// TIA Portal V20 export
// export: Created 2025-12-01T14:57:40.6788233Z, ExportSetting None, DisplayName Totally Integrated Automation Portal, DisplayVersion V20 Update 3, DisplayName TIA Portal Openness, DisplayVersion V20 Update 3, DisplayName TIA Portal Version Control Interface, DisplayVersion V20 Update 3, DisplayName STEP 7 Professional, DisplayVersion V20 Update 3, DisplayName STEP 7 Safety, DisplayVersion V20 Update 2, DisplayName WinCC Basic/Comfort/Advanced, DisplayVersion V20 Update 3, DisplayName WinCC Professional, DisplayVersion V20 Update 3, DisplayName WinCC Unified, DisplayVersion V20 Update 3
FUNCTION_BLOCK "FB291_M_CIMCORP_Descarga_Doble"   // FB291, LAD
TITLE = M_TRANSLO_CS_DESCARGA_E0_S3
{ S7_Optimized_Access := 'FALSE' }
AUTHOR : CIMCORP
NAME : 20160509
VERSION : 3.4
// stored: AutoNumber false, SetENOAutomatically false
   VAR_INPUT
      Mesa : UInt;   // Mesa de la FB
      Error_Tx : Bool;   // Error en el Tx
      EnTension : Bool;   // Existe Tension en la Mesa
      Termico_Tx : Bool;   // Proteccion del Tx
      pHsMx_P1 : Bool;   // pHs 1 de la Mesa
      pHsMx_P2 : Bool;   // pHs 2 de la Mesa
      pHsMx_Seg : Bool;   // pHs Seguridad de la Mesa
      Avance_Tx : Bool;   // Avance del Tx
      CIMCORP_MoveOK_P1 : Bool;   // CIMCORP >> Move OK P01
      CIMCORP_MoveOK_P2 : Bool;   // CIMCORP >> Move OK P02
      CIMCORP_Stop : Bool;   // CIMCORP >> Stop
      PTF_Mx_MSig : Bool;   // S3 >> Mesa Siguiente PTF
      FTF_Mx_MSig : Bool;   // S3 >> Mesa Siguiente FTF
      MSig_CargaAct : Bool;
      Mx_VelocidadLenta_In : Bool;   // Forzar a Velociada Lenta
      F_EnvMens_Mx : Bool;   // Fin de Envio de Mensaje
      OrdSal_S03 : Bool;   // Orden de Salida por S3
      V_CNT_ApHsMx : Int := 200;   // Valor de Ausencia
      V_CNTSeg_ApHsMx : Int := 2000;   // Valor de Seguriadad para Ausencia
      V_CNT_PerdidapHs : Int := 1000;   // CNT de Perdida de pHs
   END_VAR
   VAR_OUTPUT
      P_EnvMens_PMx : Bool;   // Permiso de Enviar Mensaje de Presencia
      P_RecepOK_Mx : Bool;   // Recepcion OK
      AVTF_Mx_MSig : Bool;   // S3 >> Mesa Siguiente AVTF
      P_Mens_Mx_MSig : Bool;   // S3 >> Mesa Siguiente P_Mens
   END_VAR
   VAR
      Mx_ET00 : Bool;
      Mx_ET01 : Bool;
      Mx_ET02 : Bool;
      Mx_ET06 : Bool;
      Mx_ET07 : Bool;
      Mx_ET08 : Bool;
      Mx_ET09 : Bool;
      Mx_ET10 : Bool;
      Mx_ET11 : Bool;
      Mx_ET110 : Bool;
      Mx_ET111 : Bool;
      Mx_ET20 : Bool;
      Mx_ET21 : Bool;
      Mx_ET120 : Bool;
      Mx_ET121 : Bool;
      Mx_ET50 : Bool;
      Mx_ET51 : Bool;
      Mx_ET150 : Bool;
      Mx_ET151 : Bool;
      CIMCORP_OK : Bool;   // CIMCORP >> Esta En Marcha
      CNT_ApHsMx { S7_SetPoint := 'True'} : "FB910_CNT_UHS";   // CNT de la Ausencia
      CNTSeg_ApHsMx { S7_SetPoint := 'True'} : "FB910_CNT_UHS";   // CNT de Seguridad de la Ausencia
      TMP_EnTension { S7_SetPoint := 'True'} : "FB910_CNT_UHS";
      CNT_PerdidapHs { S7_SetPoint := 'True'} : "FB910_CNT_UHS";   // CNT de Perdida de pHs
      STAT_EnvMens_PMx : Bool;   // Interna >> Envio del Mensaje de Presencia
      STAT_AVTF_Mx_MSig : Bool;   // Interna >> AVTF de Mx >> MSig
      MA_UnLoadOK_P1 : Bool;
      MA_UnLoadOK_P2 : Bool;
   END_VAR
   VAR_TEMP
      EstadoZona : "EstadoZona";   // Estado de Zona de la Mesa
      EstadoVI : "EstadosMesa";   // Estado del Vehiculo Inteliguente de la Mesa
      ConfigFB : "UDT_ConfigFB";   // Configuracion de la FB de la Mesa
      Aux_ET00 : Bool;
   END_VAR
BEGIN

REGION Network 1: INICIALIZAR - Recoger las Variables de Estado de la Mesa
   // Se recoge - Estado_CBx
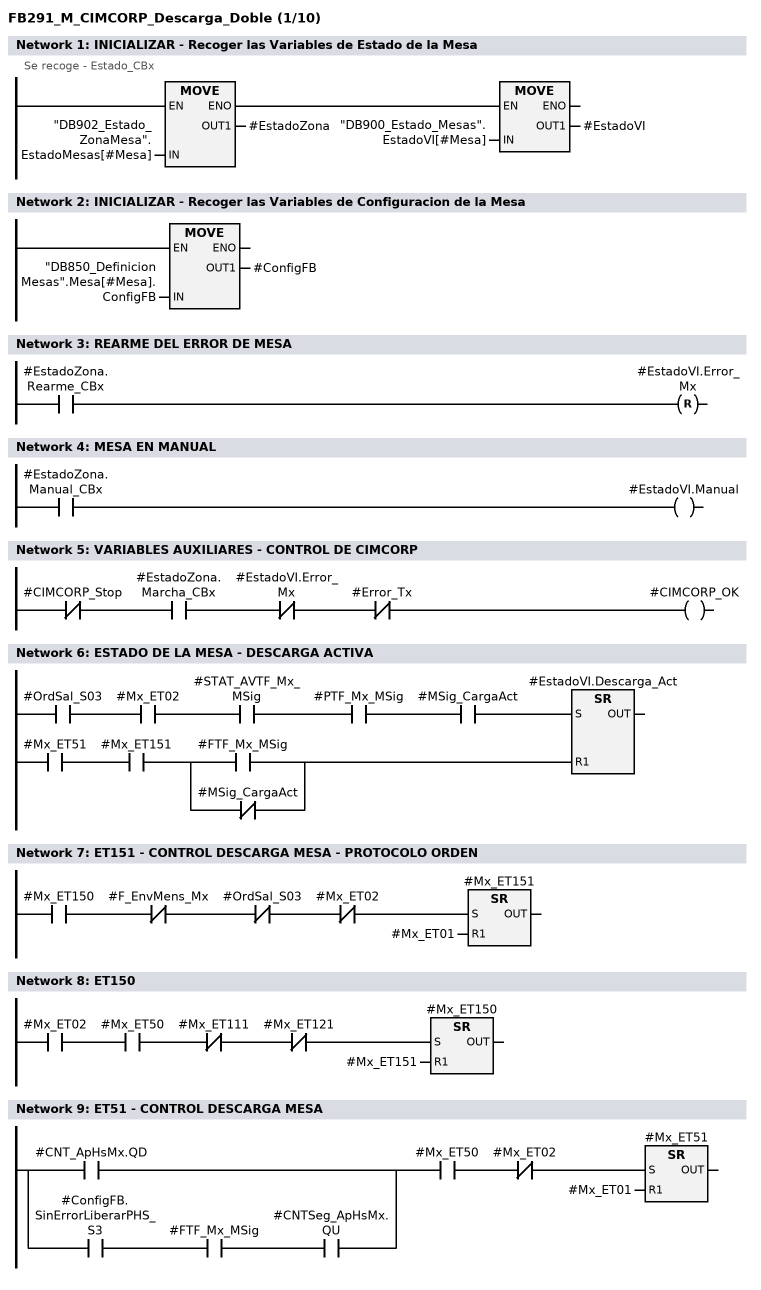
   RUNG wire#powerrail
      Move(in := "DB902_Estado_ZonaMesa".EstadoMesas[#Mesa], out1 => #EstadoZona)
      Move(in := "DB900_Estado_Mesas".EstadoVI[#Mesa], out1 => #EstadoVI)
   END_RUNG
   // the same network as SCL:
   #EstadoZona := "DB902_Estado_ZonaMesa".EstadoMesas[#Mesa];
   #EstadoVI := "DB900_Estado_Mesas".EstadoVI[#Mesa];
END_REGION

REGION Network 2: INICIALIZAR - Recoger las Variables de Configuracion de la Mesa
   RUNG wire#powerrail
      Move(in := "DB850_DefinicionMesas".Mesa[#Mesa].ConfigFB, out1 => #ConfigFB)
   END_RUNG
   // the same network as SCL:
   #ConfigFB := "DB850_DefinicionMesas".Mesa[#Mesa].ConfigFB;
END_REGION

REGION Network 3: REARME DEL ERROR DE MESA
   RUNG wire#powerrail
      Contact( #EstadoZona.Rearme_CBx )
      R_Coil( #EstadoVI.Error_Mx )
   END_RUNG
   // the same network as SCL:
   IF #EstadoZona.Rearme_CBx THEN #EstadoVI.Error_Mx := FALSE; END_IF;
END_REGION

REGION Network 4: MESA EN MANUAL
   RUNG wire#powerrail
      Contact( #EstadoZona.Manual_CBx )
      Coil( #EstadoVI.Manual )
   END_RUNG
   // the same network as SCL:
   #EstadoVI.Manual := #EstadoZona.Manual_CBx;
END_REGION

REGION Network 5: VARIABLES AUXILIARES - CONTROL DE CIMCORP
   RUNG wire#powerrail
      I_Contact( #CIMCORP_Stop )
      Contact( #EstadoZona.Marcha_CBx )
      I_Contact( #EstadoVI.Error_Mx )
      I_Contact( #Error_Tx )
      Coil( #CIMCORP_OK )
   END_RUNG
   // the same network as SCL:
   #CIMCORP_OK := NOT #CIMCORP_Stop AND #EstadoZona.Marcha_CBx AND NOT #EstadoVI.Error_Mx AND NOT #Error_Tx;
END_REGION

REGION Network 6: ESTADO DE LA MESA - DESCARGA ACTIVA
   RUNG wire#powerrail
      Contact( #OrdSal_S03 )
      Contact( #Mx_ET02 )
      Contact( #STAT_AVTF_Mx_MSig )
      Contact( #PTF_Mx_MSig )
      Contact( #MSig_CargaAct )
      S_SR(operand := #EstadoVI.Descarga_Act, r1 := wire#w2)
   END_RUNG
   RUNG wire#powerrail
      Contact( #Mx_ET51 )
      Contact( #Mx_ET151 )
      wire#w1
      Contact( #FTF_Mx_MSig )
   END_RUNG wire#w2
   RUNG wire#w1
      I_Contact( #MSig_CargaAct )
   END_RUNG wire#w2
   // the same network as SCL:
   IF #OrdSal_S03 AND #Mx_ET02 AND #STAT_AVTF_Mx_MSig AND #PTF_Mx_MSig AND #MSig_CargaAct THEN
       #EstadoVI.Descarga_Act := TRUE;   // SR flip-flop
   END_IF;
   IF #Mx_ET51 AND #Mx_ET151 AND (#FTF_Mx_MSig OR NOT #MSig_CargaAct) THEN
       #EstadoVI.Descarga_Act := FALSE;
   END_IF;
END_REGION

REGION Network 7: ET151 - CONTROL DESCARGA MESA - PROTOCOLO ORDEN
   RUNG wire#powerrail
      Contact( #Mx_ET150 )
      I_Contact( #F_EnvMens_Mx )
      I_Contact( #OrdSal_S03 )
      I_Contact( #Mx_ET02 )
      S_SR(operand := #Mx_ET151, r1 := #Mx_ET01)
   END_RUNG
   // the same network as SCL:
   IF #Mx_ET150 AND NOT #F_EnvMens_Mx AND NOT #OrdSal_S03 AND NOT #Mx_ET02 THEN
       #Mx_ET151 := TRUE;   // SR flip-flop
   END_IF;
   IF #Mx_ET01 THEN #Mx_ET151 := FALSE; END_IF;
END_REGION

REGION Network 8: ET150
   RUNG wire#powerrail
      Contact( #Mx_ET02 )
      Contact( #Mx_ET50 )
      I_Contact( #Mx_ET111 )
      I_Contact( #Mx_ET121 )
      S_SR(operand := #Mx_ET150, r1 := #Mx_ET151)
   END_RUNG
   // the same network as SCL:
   IF #Mx_ET02 AND #Mx_ET50 AND NOT #Mx_ET111 AND NOT #Mx_ET121 THEN
       #Mx_ET150 := TRUE;   // SR flip-flop
   END_IF;
   IF #Mx_ET151 THEN #Mx_ET150 := FALSE; END_IF;
END_REGION

REGION Network 9: ET51 - CONTROL DESCARGA MESA
   RUNG wire#powerrail
      Contact( #CNT_ApHsMx.QD )
      wire#w1
      Contact( #Mx_ET50 )
      I_Contact( #Mx_ET02 )
      S_SR(operand := #Mx_ET51, r1 := #Mx_ET01)
   END_RUNG
   RUNG wire#powerrail
      Contact( #ConfigFB.SinErrorLiberarPHS_S3 )
      Contact( #FTF_Mx_MSig )
      Contact( #CNTSeg_ApHsMx.QU )
   END_RUNG wire#w1
   // the same network as SCL:
   IF (#CNT_ApHsMx.QD OR (#ConfigFB.SinErrorLiberarPHS_S3 AND #FTF_Mx_MSig AND #CNTSeg_ApHsMx.QU)) AND #Mx_ET50 AND NOT #Mx_ET02 THEN
       #Mx_ET51 := TRUE;   // SR flip-flop
   END_IF;
   IF #Mx_ET01 THEN #Mx_ET51 := FALSE; END_IF;
END_REGION

REGION Network 10: ET50
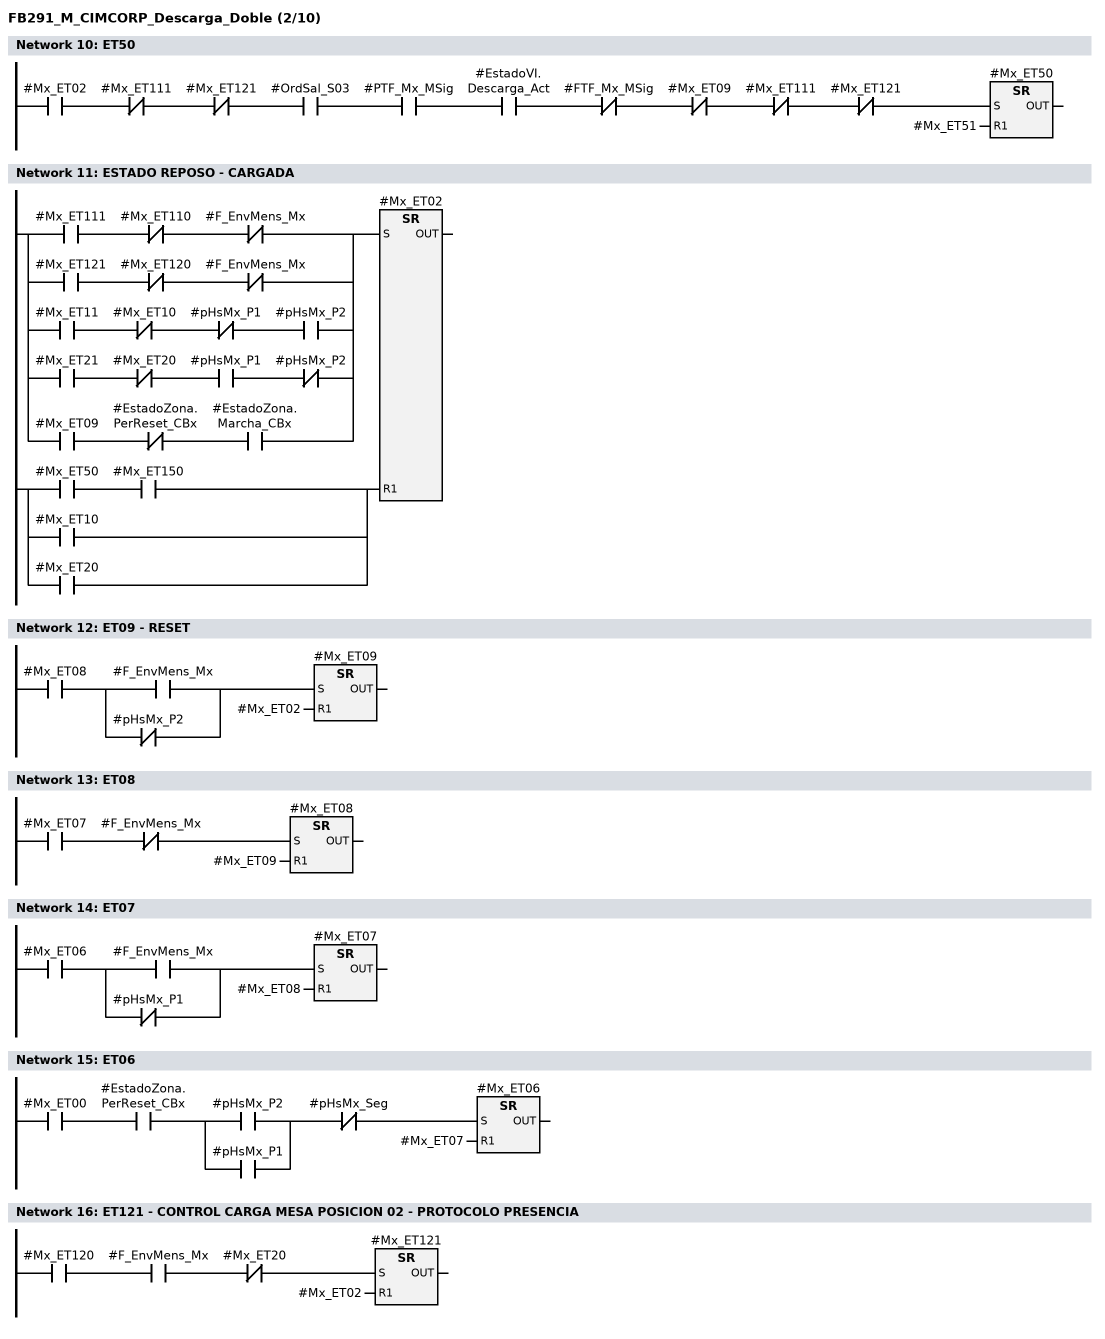
   RUNG wire#powerrail
      Contact( #Mx_ET02 )
      I_Contact( #Mx_ET111 )
      I_Contact( #Mx_ET121 )
      Contact( #OrdSal_S03 )
      Contact( #PTF_Mx_MSig )
      Contact( #EstadoVI.Descarga_Act )
      I_Contact( #FTF_Mx_MSig )
      I_Contact( #Mx_ET09 )
      I_Contact( #Mx_ET111 )
      I_Contact( #Mx_ET121 )
      S_SR(operand := #Mx_ET50, r1 := #Mx_ET51)
   END_RUNG
   // the same network as SCL:
   IF #Mx_ET02 AND NOT #Mx_ET111 AND NOT #Mx_ET121 AND #OrdSal_S03 AND #PTF_Mx_MSig AND #EstadoVI.Descarga_Act AND NOT #FTF_Mx_MSig AND NOT #Mx_ET09 AND NOT #Mx_ET111 AND NOT #Mx_ET121 THEN
       #Mx_ET50 := TRUE;   // SR flip-flop
   END_IF;
   IF #Mx_ET51 THEN #Mx_ET50 := FALSE; END_IF;
END_REGION

REGION Network 11: ESTADO REPOSO - CARGADA
   RUNG wire#powerrail
      Contact( #Mx_ET111 )
      I_Contact( #Mx_ET110 )
      I_Contact( #F_EnvMens_Mx )
      wire#w1
      S_SR(operand := #Mx_ET02, r1 := wire#w2)
   END_RUNG
   RUNG wire#powerrail
      Contact( #Mx_ET121 )
      I_Contact( #Mx_ET120 )
      I_Contact( #F_EnvMens_Mx )
   END_RUNG wire#w1
   RUNG wire#powerrail
      Contact( #Mx_ET11 )
      I_Contact( #Mx_ET10 )
      I_Contact( #pHsMx_P1 )
      Contact( #pHsMx_P2 )
   END_RUNG wire#w1
   RUNG wire#powerrail
      Contact( #Mx_ET21 )
      I_Contact( #Mx_ET20 )
      Contact( #pHsMx_P1 )
      I_Contact( #pHsMx_P2 )
   END_RUNG wire#w1
   RUNG wire#powerrail
      Contact( #Mx_ET09 )
      I_Contact( #EstadoZona.PerReset_CBx )
      Contact( #EstadoZona.Marcha_CBx )
   END_RUNG wire#w1
   RUNG wire#powerrail
      Contact( #Mx_ET50 )
      Contact( #Mx_ET150 )
   END_RUNG wire#w2
   RUNG wire#powerrail
      Contact( #Mx_ET10 )
   END_RUNG wire#w2
   RUNG wire#powerrail
      Contact( #Mx_ET20 )
   END_RUNG wire#w2
   // the same network as SCL:
   IF (#Mx_ET111 AND NOT #Mx_ET110 AND NOT #F_EnvMens_Mx) OR (#Mx_ET121 AND NOT #Mx_ET120 AND NOT #F_EnvMens_Mx) OR (#Mx_ET11 AND NOT #Mx_ET10 AND NOT #pHsMx_P1 AND #pHsMx_P2) OR (#Mx_ET21 AND NOT #Mx_ET20 AND #pHsMx_P1 AND NOT #pHsMx_P2) OR (#Mx_ET09 AND NOT #EstadoZona.PerReset_CBx AND #EstadoZona.Marcha_CBx) THEN
       #Mx_ET02 := TRUE;   // SR flip-flop
   END_IF;
   IF (#Mx_ET50 AND #Mx_ET150) OR #Mx_ET10 OR #Mx_ET20 THEN #Mx_ET02 := FALSE; END_IF;
END_REGION

REGION Network 12: ET09 - RESET
   RUNG wire#powerrail
      Contact( #Mx_ET08 )
      wire#w1
      Contact( #F_EnvMens_Mx )
      wire#w2
      S_SR(operand := #Mx_ET09, r1 := #Mx_ET02)
   END_RUNG
   RUNG wire#w1
      I_Contact( #pHsMx_P2 )
   END_RUNG wire#w2
   // the same network as SCL:
   IF #Mx_ET08 AND (#F_EnvMens_Mx OR NOT #pHsMx_P2) THEN
       #Mx_ET09 := TRUE;   // SR flip-flop
   END_IF;
   IF #Mx_ET02 THEN #Mx_ET09 := FALSE; END_IF;
END_REGION

REGION Network 13: ET08
   RUNG wire#powerrail
      Contact( #Mx_ET07 )
      I_Contact( #F_EnvMens_Mx )
      S_SR(operand := #Mx_ET08, r1 := #Mx_ET09)
   END_RUNG
   // the same network as SCL:
   IF #Mx_ET07 AND NOT #F_EnvMens_Mx THEN
       #Mx_ET08 := TRUE;   // SR flip-flop
   END_IF;
   IF #Mx_ET09 THEN #Mx_ET08 := FALSE; END_IF;
END_REGION

REGION Network 14: ET07
   RUNG wire#powerrail
      Contact( #Mx_ET06 )
      wire#w1
      Contact( #F_EnvMens_Mx )
      wire#w2
      S_SR(operand := #Mx_ET07, r1 := #Mx_ET08)
   END_RUNG
   RUNG wire#w1
      I_Contact( #pHsMx_P1 )
   END_RUNG wire#w2
   // the same network as SCL:
   IF #Mx_ET06 AND (#F_EnvMens_Mx OR NOT #pHsMx_P1) THEN
       #Mx_ET07 := TRUE;   // SR flip-flop
   END_IF;
   IF #Mx_ET08 THEN #Mx_ET07 := FALSE; END_IF;
END_REGION

REGION Network 15: ET06
   RUNG wire#powerrail
      Contact( #Mx_ET00 )
      Contact( #EstadoZona.PerReset_CBx )
      wire#w1
      Contact( #pHsMx_P2 )
      wire#w2
      I_Contact( #pHsMx_Seg )
      S_SR(operand := #Mx_ET06, r1 := #Mx_ET07)
   END_RUNG
   RUNG wire#w1
      Contact( #pHsMx_P1 )
   END_RUNG wire#w2
   // the same network as SCL:
   IF #Mx_ET00 AND #EstadoZona.PerReset_CBx AND (#pHsMx_P2 OR #pHsMx_P1) AND NOT #pHsMx_Seg THEN
       #Mx_ET06 := TRUE;   // SR flip-flop
   END_IF;
   IF #Mx_ET07 THEN #Mx_ET06 := FALSE; END_IF;
END_REGION

REGION Network 16: ET121 - CONTROL CARGA MESA POSICION 02 - PROTOCOLO PRESENCIA
   RUNG wire#powerrail
      Contact( #Mx_ET120 )
      Contact( #F_EnvMens_Mx )
      I_Contact( #Mx_ET20 )
      S_SR(operand := #Mx_ET121, r1 := #Mx_ET02)
   END_RUNG
   // the same network as SCL:
   IF #Mx_ET120 AND #F_EnvMens_Mx AND NOT #Mx_ET20 THEN
       #Mx_ET121 := TRUE;   // SR flip-flop
   END_IF;
   IF #Mx_ET02 THEN #Mx_ET121 := FALSE; END_IF;
END_REGION

REGION Network 17: ET120
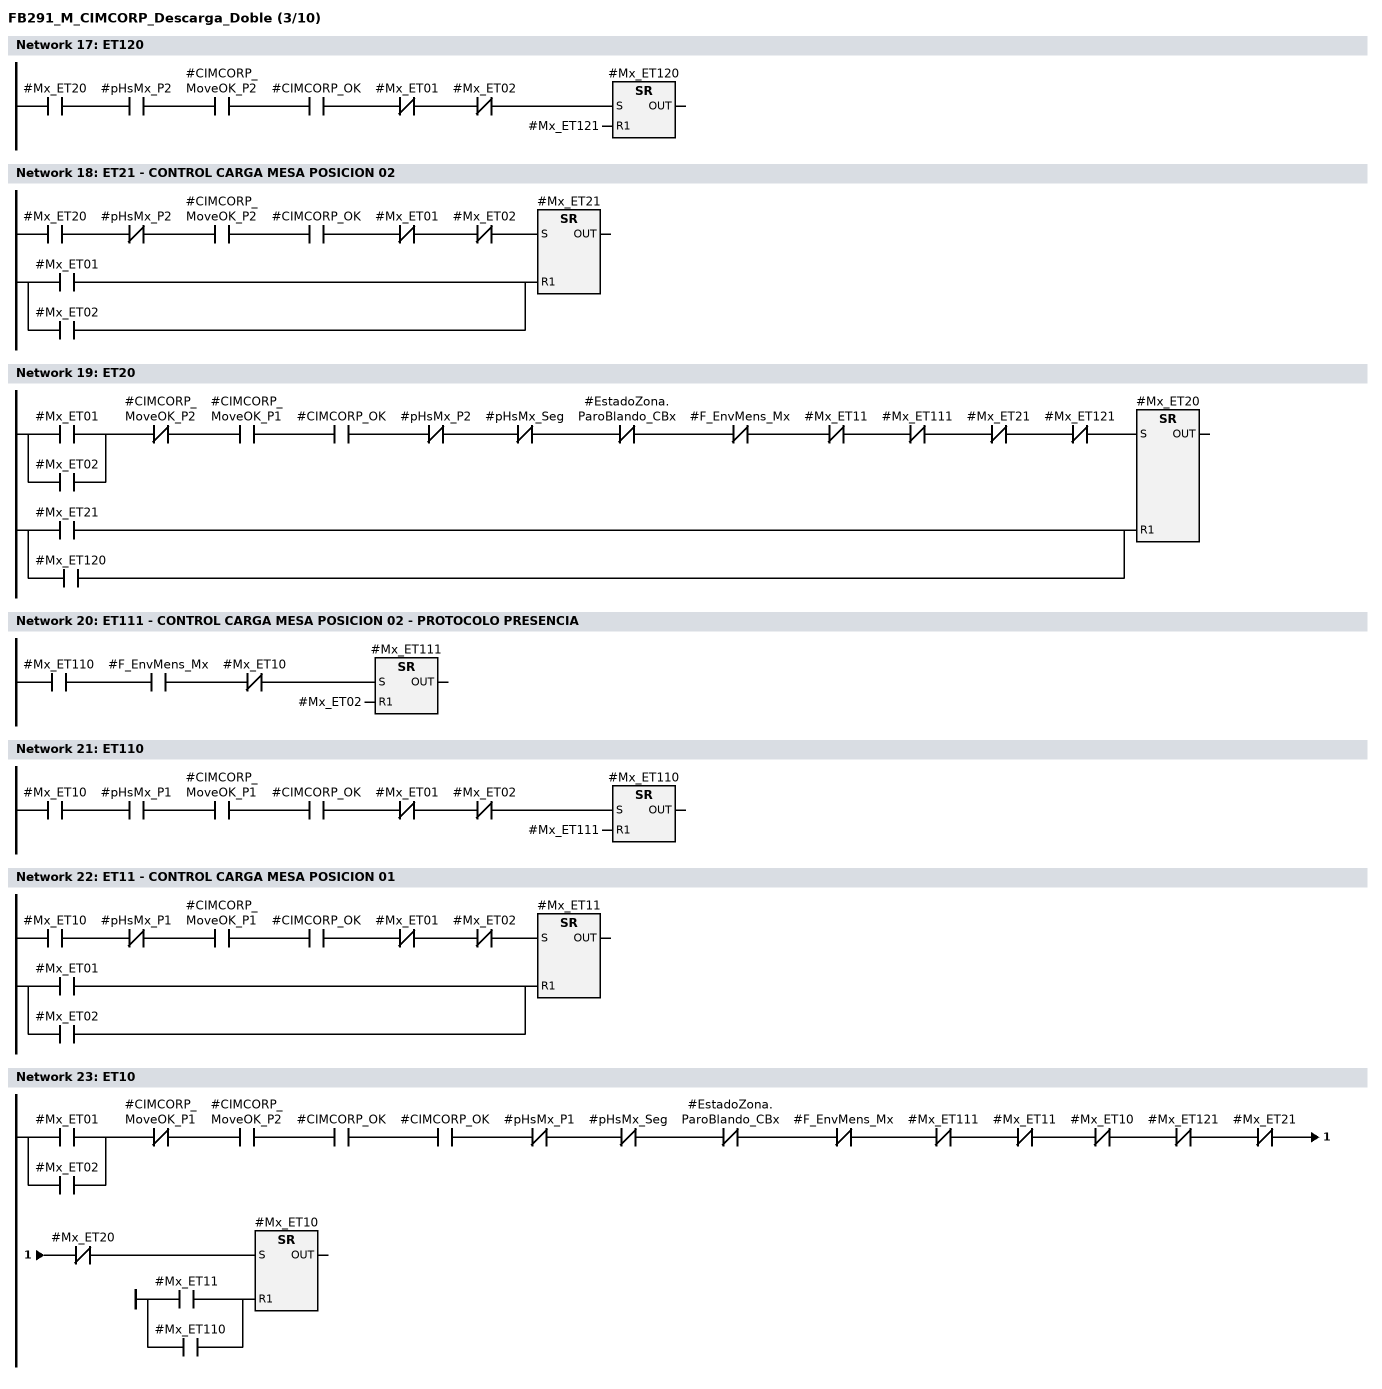
   RUNG wire#powerrail
      Contact( #Mx_ET20 )
      Contact( #pHsMx_P2 )
      Contact( #CIMCORP_MoveOK_P2 )
      Contact( #CIMCORP_OK )
      I_Contact( #Mx_ET01 )
      I_Contact( #Mx_ET02 )
      S_SR(operand := #Mx_ET120, r1 := #Mx_ET121)
   END_RUNG
   // the same network as SCL:
   IF #Mx_ET20 AND #pHsMx_P2 AND #CIMCORP_MoveOK_P2 AND #CIMCORP_OK AND NOT #Mx_ET01 AND NOT #Mx_ET02 THEN
       #Mx_ET120 := TRUE;   // SR flip-flop
   END_IF;
   IF #Mx_ET121 THEN #Mx_ET120 := FALSE; END_IF;
END_REGION

REGION Network 18: ET21 - CONTROL CARGA MESA POSICION 02
   RUNG wire#powerrail
      Contact( #Mx_ET20 )
      I_Contact( #pHsMx_P2 )
      Contact( #CIMCORP_MoveOK_P2 )
      Contact( #CIMCORP_OK )
      I_Contact( #Mx_ET01 )
      I_Contact( #Mx_ET02 )
      S_SR(operand := #Mx_ET21, r1 := wire#w1)
   END_RUNG
   RUNG wire#powerrail
      Contact( #Mx_ET01 )
   END_RUNG wire#w1
   RUNG wire#powerrail
      Contact( #Mx_ET02 )
   END_RUNG wire#w1
   // the same network as SCL:
   IF #Mx_ET20 AND NOT #pHsMx_P2 AND #CIMCORP_MoveOK_P2 AND #CIMCORP_OK AND NOT #Mx_ET01 AND NOT #Mx_ET02 THEN
       #Mx_ET21 := TRUE;   // SR flip-flop
   END_IF;
   IF #Mx_ET01 OR #Mx_ET02 THEN #Mx_ET21 := FALSE; END_IF;
END_REGION

REGION Network 19: ET20
   RUNG wire#powerrail
      Contact( #Mx_ET01 )
      wire#w1
      I_Contact( #CIMCORP_MoveOK_P2 )
      Contact( #CIMCORP_MoveOK_P1 )
      Contact( #CIMCORP_OK )
      I_Contact( #pHsMx_P2 )
      I_Contact( #pHsMx_Seg )
      I_Contact( #EstadoZona.ParoBlando_CBx )
      I_Contact( #F_EnvMens_Mx )
      I_Contact( #Mx_ET11 )
      I_Contact( #Mx_ET111 )
      I_Contact( #Mx_ET21 )
      I_Contact( #Mx_ET121 )
      S_SR(operand := #Mx_ET20, r1 := wire#w2)
   END_RUNG
   RUNG wire#powerrail
      Contact( #Mx_ET02 )
   END_RUNG wire#w1
   RUNG wire#powerrail
      Contact( #Mx_ET21 )
   END_RUNG wire#w2
   RUNG wire#powerrail
      Contact( #Mx_ET120 )
   END_RUNG wire#w2
   // the same network as SCL:
   IF (#Mx_ET01 OR #Mx_ET02) AND NOT #CIMCORP_MoveOK_P2 AND #CIMCORP_MoveOK_P1 AND #CIMCORP_OK AND NOT #pHsMx_P2 AND NOT #pHsMx_Seg AND NOT #EstadoZona.ParoBlando_CBx AND NOT #F_EnvMens_Mx AND NOT #Mx_ET11 AND NOT #Mx_ET111 AND NOT #Mx_ET21 AND NOT #Mx_ET121 THEN
       #Mx_ET20 := TRUE;   // SR flip-flop
   END_IF;
   IF #Mx_ET21 OR #Mx_ET120 THEN #Mx_ET20 := FALSE; END_IF;
END_REGION

REGION Network 20: ET111 - CONTROL CARGA MESA POSICION 02 - PROTOCOLO PRESENCIA
   RUNG wire#powerrail
      Contact( #Mx_ET110 )
      Contact( #F_EnvMens_Mx )
      I_Contact( #Mx_ET10 )
      S_SR(operand := #Mx_ET111, r1 := #Mx_ET02)
   END_RUNG
   // the same network as SCL:
   IF #Mx_ET110 AND #F_EnvMens_Mx AND NOT #Mx_ET10 THEN
       #Mx_ET111 := TRUE;   // SR flip-flop
   END_IF;
   IF #Mx_ET02 THEN #Mx_ET111 := FALSE; END_IF;
END_REGION

REGION Network 21: ET110
   RUNG wire#powerrail
      Contact( #Mx_ET10 )
      Contact( #pHsMx_P1 )
      Contact( #CIMCORP_MoveOK_P1 )
      Contact( #CIMCORP_OK )
      I_Contact( #Mx_ET01 )
      I_Contact( #Mx_ET02 )
      S_SR(operand := #Mx_ET110, r1 := #Mx_ET111)
   END_RUNG
   // the same network as SCL:
   IF #Mx_ET10 AND #pHsMx_P1 AND #CIMCORP_MoveOK_P1 AND #CIMCORP_OK AND NOT #Mx_ET01 AND NOT #Mx_ET02 THEN
       #Mx_ET110 := TRUE;   // SR flip-flop
   END_IF;
   IF #Mx_ET111 THEN #Mx_ET110 := FALSE; END_IF;
END_REGION

REGION Network 22: ET11 - CONTROL CARGA MESA POSICION 01
   RUNG wire#powerrail
      Contact( #Mx_ET10 )
      I_Contact( #pHsMx_P1 )
      Contact( #CIMCORP_MoveOK_P1 )
      Contact( #CIMCORP_OK )
      I_Contact( #Mx_ET01 )
      I_Contact( #Mx_ET02 )
      S_SR(operand := #Mx_ET11, r1 := wire#w1)
   END_RUNG
   RUNG wire#powerrail
      Contact( #Mx_ET01 )
   END_RUNG wire#w1
   RUNG wire#powerrail
      Contact( #Mx_ET02 )
   END_RUNG wire#w1
   // the same network as SCL:
   IF #Mx_ET10 AND NOT #pHsMx_P1 AND #CIMCORP_MoveOK_P1 AND #CIMCORP_OK AND NOT #Mx_ET01 AND NOT #Mx_ET02 THEN
       #Mx_ET11 := TRUE;   // SR flip-flop
   END_IF;
   IF #Mx_ET01 OR #Mx_ET02 THEN #Mx_ET11 := FALSE; END_IF;
END_REGION

REGION Network 23: ET10
   RUNG wire#powerrail
      Contact( #Mx_ET01 )
      wire#w1
      I_Contact( #CIMCORP_MoveOK_P1 )
      Contact( #CIMCORP_MoveOK_P2 )
      Contact( #CIMCORP_OK )
      Contact( #CIMCORP_OK )
      I_Contact( #pHsMx_P1 )
      I_Contact( #pHsMx_Seg )
      I_Contact( #EstadoZona.ParoBlando_CBx )
      I_Contact( #F_EnvMens_Mx )
      I_Contact( #Mx_ET111 )
      I_Contact( #Mx_ET11 )
      I_Contact( #Mx_ET10 )
      I_Contact( #Mx_ET121 )
      I_Contact( #Mx_ET21 )
      I_Contact( #Mx_ET20 )
      S_SR(operand := #Mx_ET10, r1 := wire#w2)
   END_RUNG
   RUNG wire#powerrail
      Contact( #Mx_ET02 )
   END_RUNG wire#w1
   RUNG wire#powerrail
      Contact( #Mx_ET11 )
   END_RUNG wire#w2
   RUNG wire#powerrail
      Contact( #Mx_ET110 )
   END_RUNG wire#w2
   // the same network as SCL:
   IF (#Mx_ET01 OR #Mx_ET02) AND NOT #CIMCORP_MoveOK_P1 AND #CIMCORP_MoveOK_P2 AND #CIMCORP_OK AND #CIMCORP_OK AND NOT #pHsMx_P1 AND NOT #pHsMx_Seg AND NOT #EstadoZona.ParoBlando_CBx AND NOT #F_EnvMens_Mx AND NOT #Mx_ET111 AND NOT #Mx_ET11 AND NOT #Mx_ET10 AND NOT #Mx_ET121 AND NOT #Mx_ET21 AND NOT #Mx_ET20 THEN
       #Mx_ET10 := TRUE;   // SR flip-flop
   END_IF;
   IF #Mx_ET11 OR #Mx_ET110 THEN #Mx_ET10 := FALSE; END_IF;
END_REGION

REGION Network 24: ET01 - ESTADO REPOSO - VACIO
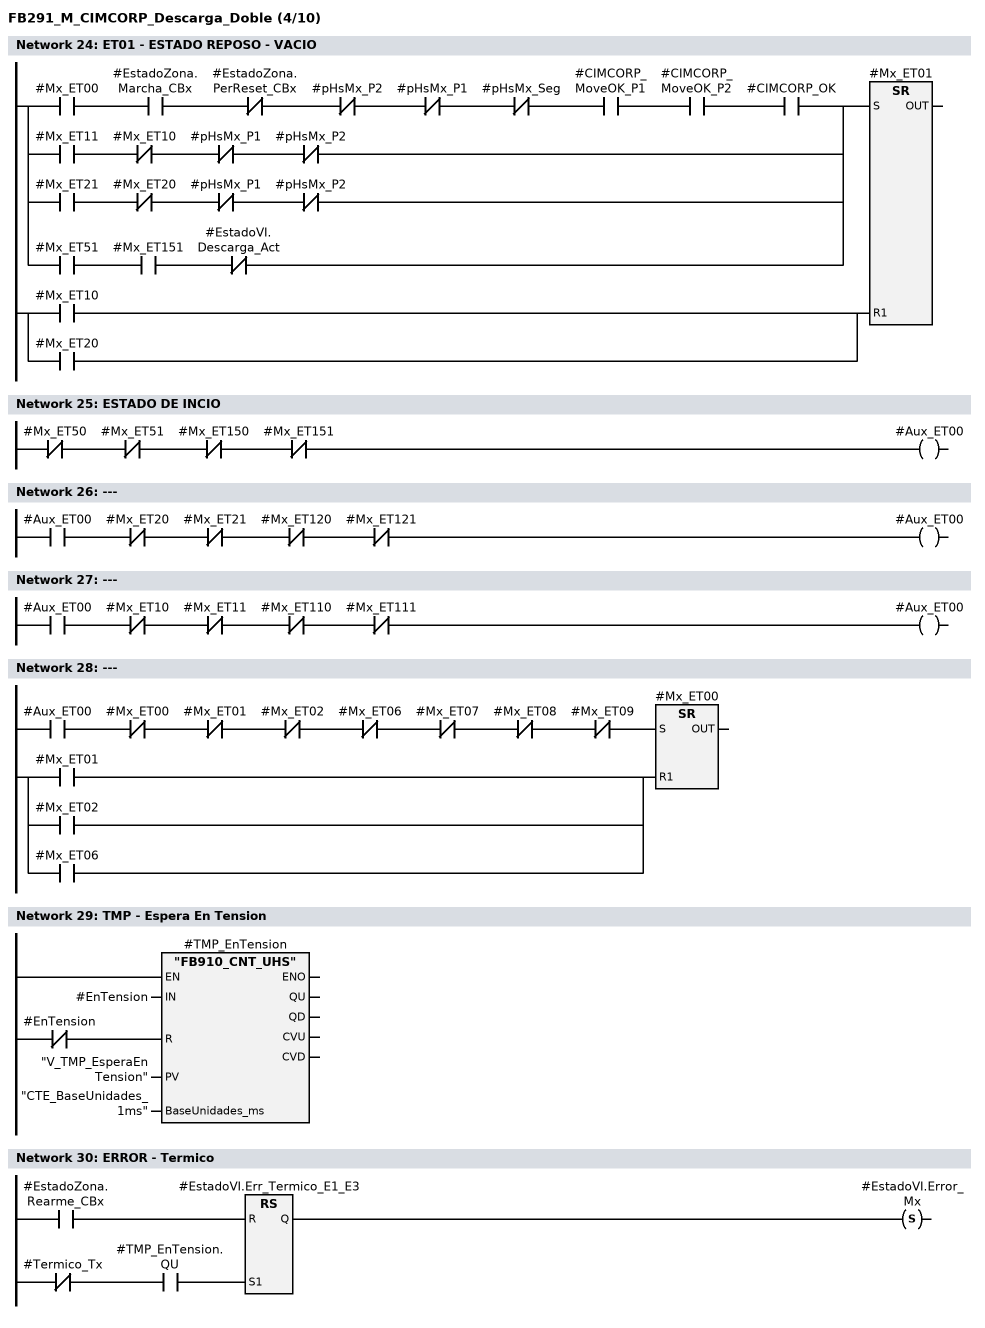
   RUNG wire#powerrail
      Contact( #Mx_ET00 )
      Contact( #EstadoZona.Marcha_CBx )
      I_Contact( #EstadoZona.PerReset_CBx )
      I_Contact( #pHsMx_P2 )
      I_Contact( #pHsMx_P1 )
      I_Contact( #pHsMx_Seg )
      Contact( #CIMCORP_MoveOK_P1 )
      Contact( #CIMCORP_MoveOK_P2 )
      Contact( #CIMCORP_OK )
      wire#w1
      S_SR(operand := #Mx_ET01, r1 := wire#w2)
   END_RUNG
   RUNG wire#powerrail
      Contact( #Mx_ET11 )
      I_Contact( #Mx_ET10 )
      I_Contact( #pHsMx_P1 )
      I_Contact( #pHsMx_P2 )
   END_RUNG wire#w1
   RUNG wire#powerrail
      Contact( #Mx_ET21 )
      I_Contact( #Mx_ET20 )
      I_Contact( #pHsMx_P1 )
      I_Contact( #pHsMx_P2 )
   END_RUNG wire#w1
   RUNG wire#powerrail
      Contact( #Mx_ET51 )
      Contact( #Mx_ET151 )
      I_Contact( #EstadoVI.Descarga_Act )
   END_RUNG wire#w1
   RUNG wire#powerrail
      Contact( #Mx_ET10 )
   END_RUNG wire#w2
   RUNG wire#powerrail
      Contact( #Mx_ET20 )
   END_RUNG wire#w2
   // the same network as SCL:
   IF (#Mx_ET00 AND #EstadoZona.Marcha_CBx AND NOT #EstadoZona.PerReset_CBx AND NOT #pHsMx_P2 AND NOT #pHsMx_P1 AND NOT #pHsMx_Seg AND #CIMCORP_MoveOK_P1 AND #CIMCORP_MoveOK_P2 AND #CIMCORP_OK) OR (#Mx_ET11 AND NOT #Mx_ET10 AND NOT #pHsMx_P1 AND NOT #pHsMx_P2) OR (#Mx_ET21 AND NOT #Mx_ET20 AND NOT #pHsMx_P1 AND NOT #pHsMx_P2) OR (#Mx_ET51 AND #Mx_ET151 AND NOT #EstadoVI.Descarga_Act) THEN
       #Mx_ET01 := TRUE;   // SR flip-flop
   END_IF;
   IF #Mx_ET10 OR #Mx_ET20 THEN #Mx_ET01 := FALSE; END_IF;
END_REGION

REGION Network 25: ESTADO DE INCIO
   RUNG wire#powerrail
      I_Contact( #Mx_ET50 )
      I_Contact( #Mx_ET51 )
      I_Contact( #Mx_ET150 )
      I_Contact( #Mx_ET151 )
      Coil( #Aux_ET00 )
   END_RUNG
   // the same network as SCL:
   #Aux_ET00 := NOT #Mx_ET50 AND NOT #Mx_ET51 AND NOT #Mx_ET150 AND NOT #Mx_ET151;
END_REGION

REGION Network 26: ---
   RUNG wire#powerrail
      Contact( #Aux_ET00 )
      I_Contact( #Mx_ET20 )
      I_Contact( #Mx_ET21 )
      I_Contact( #Mx_ET120 )
      I_Contact( #Mx_ET121 )
      Coil( #Aux_ET00 )
   END_RUNG
   // the same network as SCL:
   #Aux_ET00 := #Aux_ET00 AND NOT #Mx_ET20 AND NOT #Mx_ET21 AND NOT #Mx_ET120 AND NOT #Mx_ET121;
END_REGION

REGION Network 27: ---
   RUNG wire#powerrail
      Contact( #Aux_ET00 )
      I_Contact( #Mx_ET10 )
      I_Contact( #Mx_ET11 )
      I_Contact( #Mx_ET110 )
      I_Contact( #Mx_ET111 )
      Coil( #Aux_ET00 )
   END_RUNG
   // the same network as SCL:
   #Aux_ET00 := #Aux_ET00 AND NOT #Mx_ET10 AND NOT #Mx_ET11 AND NOT #Mx_ET110 AND NOT #Mx_ET111;
END_REGION

REGION Network 28: ---
   RUNG wire#powerrail
      Contact( #Aux_ET00 )
      I_Contact( #Mx_ET00 )
      I_Contact( #Mx_ET01 )
      I_Contact( #Mx_ET02 )
      I_Contact( #Mx_ET06 )
      I_Contact( #Mx_ET07 )
      I_Contact( #Mx_ET08 )
      I_Contact( #Mx_ET09 )
      S_SR(operand := #Mx_ET00, r1 := wire#w1)
   END_RUNG
   RUNG wire#powerrail
      Contact( #Mx_ET01 )
   END_RUNG wire#w1
   RUNG wire#powerrail
      Contact( #Mx_ET02 )
   END_RUNG wire#w1
   RUNG wire#powerrail
      Contact( #Mx_ET06 )
   END_RUNG wire#w1
   // the same network as SCL:
   IF #Aux_ET00 AND NOT #Mx_ET00 AND NOT #Mx_ET01 AND NOT #Mx_ET02 AND NOT #Mx_ET06 AND NOT #Mx_ET07 AND NOT #Mx_ET08 AND NOT #Mx_ET09 THEN
       #Mx_ET00 := TRUE;   // SR flip-flop
   END_IF;
   IF #Mx_ET01 OR #Mx_ET02 OR #Mx_ET06 THEN #Mx_ET00 := FALSE; END_IF;
END_REGION

REGION Network 29: TMP - Espera En Tension
   RUNG wire#powerrail
      #TMP_EnTension(R := wire#w1, IN := #EnTension, PV := "V_TMP_EsperaEnTension", BaseUnidades_ms := "CTE_BaseUnidades_1ms", QU =>, QD =>, CVU =>, CVD =>)
   END_RUNG
   RUNG wire#powerrail
      I_Contact( #EnTension )
   END_RUNG wire#w1
   // the same network as SCL:
   #TMP_EnTension(IN := #EnTension,   // "FB910_CNT_UHS"
                  R := NOT #EnTension,
                  PV := "V_TMP_EsperaEnTension",
                  BaseUnidades_ms := "CTE_BaseUnidades_1ms");
END_REGION

REGION Network 30: ERROR - Termico
   RUNG wire#powerrail
      Contact( #EstadoZona.Rearme_CBx )
      S_RS(operand := #EstadoVI.Err_Termico_E1_E3, s1 := wire#w1)
      S_Coil( #EstadoVI.Error_Mx )
   END_RUNG
   RUNG wire#powerrail
      I_Contact( #Termico_Tx )
      Contact( #TMP_EnTension.QU )
   END_RUNG wire#w1
   // the same network as SCL:
   IF #EstadoZona.Rearme_CBx THEN
       #EstadoVI.Err_Termico_E1_E3 := FALSE;   // RS flip-flop
   END_IF;
   IF NOT #Termico_Tx AND #TMP_EnTension.QU THEN #EstadoVI.Err_Termico_E1_E3 := TRUE; END_IF;
   IF #EstadoVI.Err_Termico_E1_E3 THEN #EstadoVI.Error_Mx := TRUE; END_IF;
END_REGION

REGION Network 31: ERROR - Mesa Ocupada
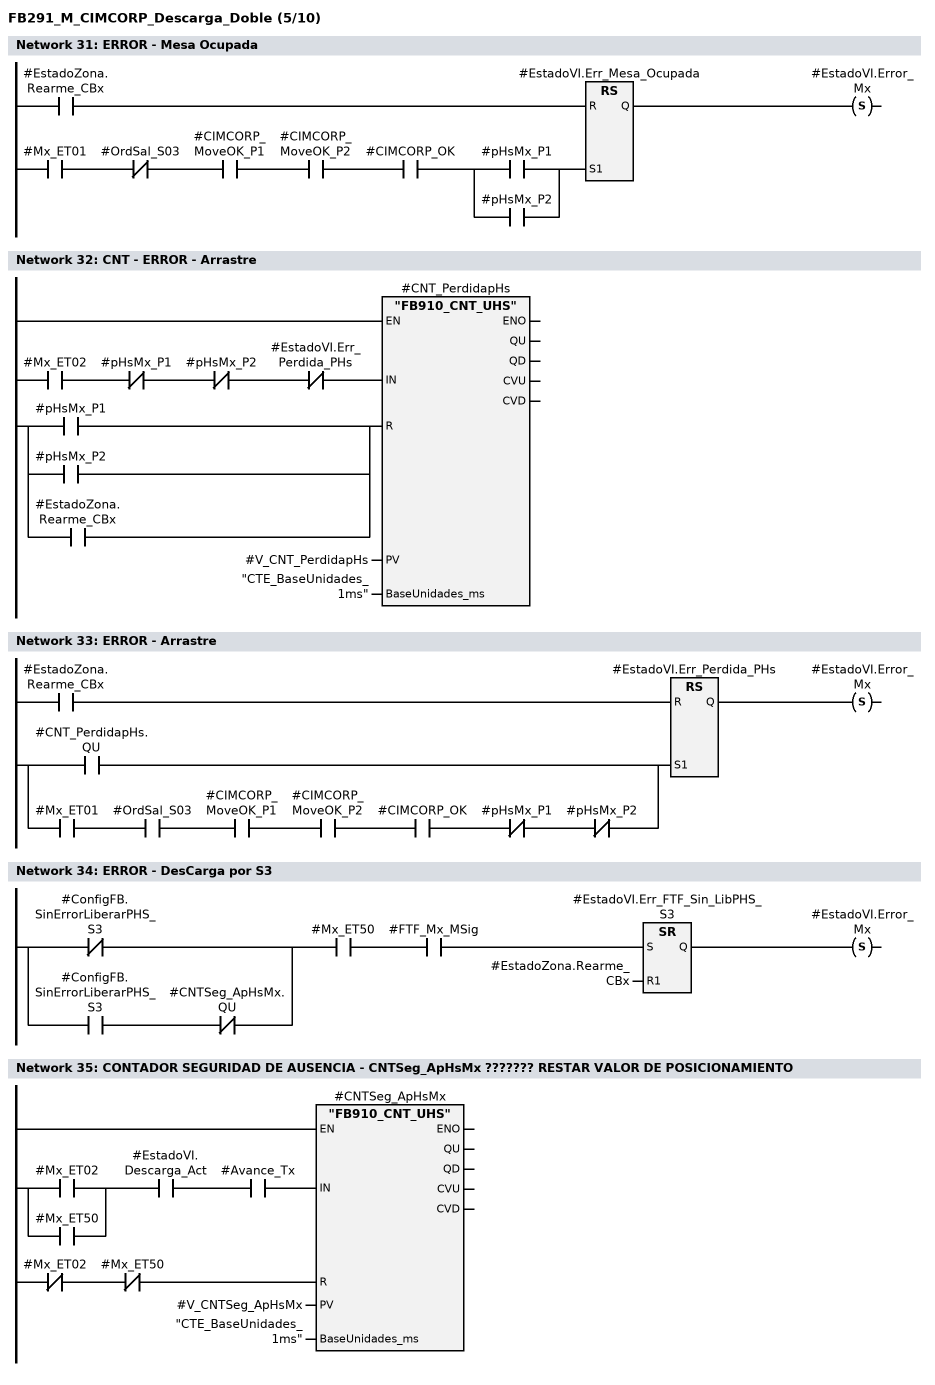
   RUNG wire#powerrail
      Contact( #EstadoZona.Rearme_CBx )
      S_RS(operand := #EstadoVI.Err_Mesa_Ocupada, s1 := wire#w2)
      S_Coil( #EstadoVI.Error_Mx )
   END_RUNG
   RUNG wire#powerrail
      Contact( #Mx_ET01 )
      I_Contact( #OrdSal_S03 )
      Contact( #CIMCORP_MoveOK_P1 )
      Contact( #CIMCORP_MoveOK_P2 )
      Contact( #CIMCORP_OK )
      wire#w1
      Contact( #pHsMx_P1 )
   END_RUNG wire#w2
   RUNG wire#w1
      Contact( #pHsMx_P2 )
   END_RUNG wire#w2
   // the same network as SCL:
   IF #EstadoZona.Rearme_CBx THEN
       #EstadoVI.Err_Mesa_Ocupada := FALSE;   // RS flip-flop
   END_IF;
   IF #Mx_ET01 AND NOT #OrdSal_S03 AND #CIMCORP_MoveOK_P1 AND #CIMCORP_MoveOK_P2 AND #CIMCORP_OK AND (#pHsMx_P1 OR #pHsMx_P2) THEN
       #EstadoVI.Err_Mesa_Ocupada := TRUE;
   END_IF;
   IF #EstadoVI.Err_Mesa_Ocupada THEN #EstadoVI.Error_Mx := TRUE; END_IF;
END_REGION

REGION Network 32: CNT - ERROR - Arrastre
   RUNG wire#powerrail
      #CNT_PerdidapHs(IN := wire#w1, R := wire#w2, PV := #V_CNT_PerdidapHs, BaseUnidades_ms := "CTE_BaseUnidades_1ms", QU =>, QD =>, CVU =>, CVD =>)
   END_RUNG
   RUNG wire#powerrail
      Contact( #Mx_ET02 )
      I_Contact( #pHsMx_P1 )
      I_Contact( #pHsMx_P2 )
      I_Contact( #EstadoVI.Err_Perdida_PHs )
   END_RUNG wire#w1
   RUNG wire#powerrail
      Contact( #pHsMx_P1 )
   END_RUNG wire#w2
   RUNG wire#powerrail
      Contact( #pHsMx_P2 )
   END_RUNG wire#w2
   RUNG wire#powerrail
      Contact( #EstadoZona.Rearme_CBx )
   END_RUNG wire#w2
   // the same network as SCL:
   #CNT_PerdidapHs(IN := #Mx_ET02 AND NOT #pHsMx_P1 AND NOT #pHsMx_P2 AND NOT #EstadoVI.Err_Perdida_PHs,   // "FB910_CNT_UHS"
                   R := #pHsMx_P1 OR #pHsMx_P2 OR #EstadoZona.Rearme_CBx,
                   PV := #V_CNT_PerdidapHs,
                   BaseUnidades_ms := "CTE_BaseUnidades_1ms");
END_REGION

REGION Network 33: ERROR - Arrastre
   RUNG wire#powerrail
      Contact( #EstadoZona.Rearme_CBx )
      S_RS(operand := #EstadoVI.Err_Perdida_PHs, s1 := wire#w1)
      S_Coil( #EstadoVI.Error_Mx )
   END_RUNG
   RUNG wire#powerrail
      Contact( #CNT_PerdidapHs.QU )
   END_RUNG wire#w1
   RUNG wire#powerrail
      Contact( #Mx_ET01 )
      Contact( #OrdSal_S03 )
      Contact( #CIMCORP_MoveOK_P1 )
      Contact( #CIMCORP_MoveOK_P2 )
      Contact( #CIMCORP_OK )
      I_Contact( #pHsMx_P1 )
      I_Contact( #pHsMx_P2 )
   END_RUNG wire#w1
   // the same network as SCL:
   IF #EstadoZona.Rearme_CBx THEN
       #EstadoVI.Err_Perdida_PHs := FALSE;   // RS flip-flop
   END_IF;
   IF #CNT_PerdidapHs.QU OR (#Mx_ET01 AND #OrdSal_S03 AND #CIMCORP_MoveOK_P1 AND #CIMCORP_MoveOK_P2 AND #CIMCORP_OK AND NOT #pHsMx_P1 AND NOT #pHsMx_P2) THEN
       #EstadoVI.Err_Perdida_PHs := TRUE;
   END_IF;
   IF #EstadoVI.Err_Perdida_PHs THEN #EstadoVI.Error_Mx := TRUE; END_IF;
END_REGION

REGION Network 34: ERROR - DesCarga por S3
   RUNG wire#powerrail
      I_Contact( #ConfigFB.SinErrorLiberarPHS_S3 )
      wire#w1
      Contact( #Mx_ET50 )
      Contact( #FTF_Mx_MSig )
      S_SR(operand := #EstadoVI.Err_FTF_Sin_LibPHS_S3, r1 := #EstadoZona.Rearme_CBx)
      S_Coil( #EstadoVI.Error_Mx )
   END_RUNG
   RUNG wire#powerrail
      Contact( #ConfigFB.SinErrorLiberarPHS_S3 )
      I_Contact( #CNTSeg_ApHsMx.QU )
   END_RUNG wire#w1
   // the same network as SCL:
   IF (NOT #ConfigFB.SinErrorLiberarPHS_S3 OR (#ConfigFB.SinErrorLiberarPHS_S3 AND NOT #CNTSeg_ApHsMx.QU)) AND #Mx_ET50 AND #FTF_Mx_MSig THEN
       #EstadoVI.Err_FTF_Sin_LibPHS_S3 := TRUE;   // SR flip-flop
   END_IF;
   IF #EstadoZona.Rearme_CBx THEN #EstadoVI.Err_FTF_Sin_LibPHS_S3 := FALSE; END_IF;
   IF #EstadoVI.Err_FTF_Sin_LibPHS_S3 THEN #EstadoVI.Error_Mx := TRUE; END_IF;
END_REGION

REGION Network 35: CONTADOR SEGURIDAD DE AUSENCIA - CNTSeg_ApHsMx ??????? RESTAR VALOR DE POSICIONAMIENTO
   RUNG wire#powerrail
      #CNTSeg_ApHsMx(IN := wire#w2, R := wire#w3, PV := #V_CNTSeg_ApHsMx, BaseUnidades_ms := "CTE_BaseUnidades_1ms", QU =>, QD =>, CVU =>, CVD =>)
   END_RUNG
   RUNG wire#powerrail
      Contact( #Mx_ET02 )
      wire#w1
      Contact( #EstadoVI.Descarga_Act )
      Contact( #Avance_Tx )
   END_RUNG wire#w2
   RUNG wire#powerrail
      Contact( #Mx_ET50 )
   END_RUNG wire#w1
   RUNG wire#powerrail
      I_Contact( #Mx_ET02 )
      I_Contact( #Mx_ET50 )
   END_RUNG wire#w3
   // the same network as SCL:
   #CNTSeg_ApHsMx(IN := (#Mx_ET02 OR #Mx_ET50) AND #EstadoVI.Descarga_Act AND #Avance_Tx,   // "FB910_CNT_UHS"
                  R := NOT #Mx_ET02 AND NOT #Mx_ET50,
                  PV := #V_CNTSeg_ApHsMx,
                  BaseUnidades_ms := "CTE_BaseUnidades_1ms");
END_REGION

REGION Network 36: CONTADOR DE LA AUSENCIA - CNT_ApHsMX
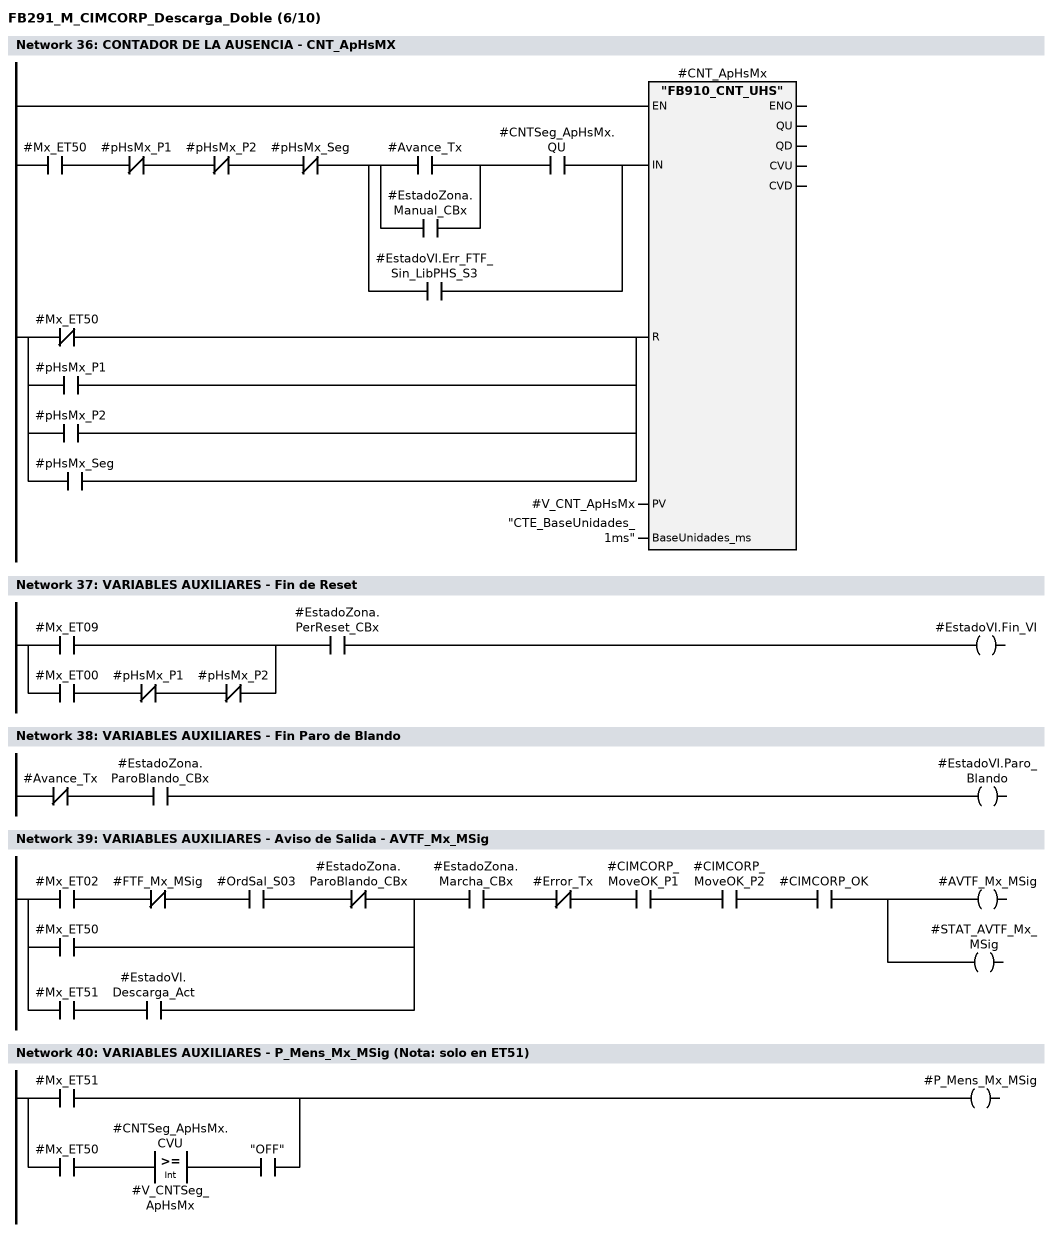
   RUNG wire#powerrail
      #CNT_ApHsMx(IN := wire#w3, R := wire#w4, PV := #V_CNT_ApHsMx, BaseUnidades_ms := "CTE_BaseUnidades_1ms", QU =>, QD =>, CVU =>, CVD =>)
   END_RUNG
   RUNG wire#powerrail
      Contact( #Mx_ET50 )
      I_Contact( #pHsMx_P1 )
      I_Contact( #pHsMx_P2 )
      I_Contact( #pHsMx_Seg )
      wire#w1
      Contact( #Avance_Tx )
      wire#w2
      Contact( #CNTSeg_ApHsMx.QU )
   END_RUNG wire#w3
   RUNG wire#w1
      Contact( #EstadoZona.Manual_CBx )
   END_RUNG wire#w2
   RUNG wire#w1
      Contact( #EstadoVI.Err_FTF_Sin_LibPHS_S3 )
   END_RUNG wire#w3
   RUNG wire#powerrail
      I_Contact( #Mx_ET50 )
   END_RUNG wire#w4
   RUNG wire#powerrail
      Contact( #pHsMx_P1 )
   END_RUNG wire#w4
   RUNG wire#powerrail
      Contact( #pHsMx_P2 )
   END_RUNG wire#w4
   RUNG wire#powerrail
      Contact( #pHsMx_Seg )
   END_RUNG wire#w4
   // the same network as SCL:
   #CNT_ApHsMx(IN := #Mx_ET50 AND NOT #pHsMx_P1 AND NOT #pHsMx_P2 AND NOT #pHsMx_Seg AND (((#Avance_Tx OR #EstadoZona.Manual_CBx) AND #CNTSeg_ApHsMx.QU) OR #EstadoVI.Err_FTF_Sin_LibPHS_S3),   // "FB910_CNT_UHS"
               R := NOT #Mx_ET50 OR #pHsMx_P1 OR #pHsMx_P2 OR #pHsMx_Seg,
               PV := #V_CNT_ApHsMx,
               BaseUnidades_ms := "CTE_BaseUnidades_1ms");
END_REGION

REGION Network 37: VARIABLES AUXILIARES - Fin de Reset
   RUNG wire#powerrail
      Contact( #Mx_ET09 )
      wire#w1
      Contact( #EstadoZona.PerReset_CBx )
      Coil( #EstadoVI.Fin_VI )
   END_RUNG
   RUNG wire#powerrail
      Contact( #Mx_ET00 )
      I_Contact( #pHsMx_P1 )
      I_Contact( #pHsMx_P2 )
   END_RUNG wire#w1
   // the same network as SCL:
   #EstadoVI.Fin_VI := (#Mx_ET09 OR (#Mx_ET00 AND NOT #pHsMx_P1 AND NOT #pHsMx_P2)) AND #EstadoZona.PerReset_CBx;
END_REGION

REGION Network 38: VARIABLES AUXILIARES - Fin Paro de Blando
   RUNG wire#powerrail
      I_Contact( #Avance_Tx )
      Contact( #EstadoZona.ParoBlando_CBx )
      Coil( #EstadoVI.Paro_Blando )
   END_RUNG
   // the same network as SCL:
   #EstadoVI.Paro_Blando := NOT #Avance_Tx AND #EstadoZona.ParoBlando_CBx;
END_REGION

REGION Network 39: VARIABLES AUXILIARES - Aviso de Salida - AVTF_Mx_MSig
   RUNG wire#powerrail
      Contact( #Mx_ET02 )
      I_Contact( #FTF_Mx_MSig )
      Contact( #OrdSal_S03 )
      I_Contact( #EstadoZona.ParoBlando_CBx )
      wire#w1
      Contact( #EstadoZona.Marcha_CBx )
      I_Contact( #Error_Tx )
      Contact( #CIMCORP_MoveOK_P1 )
      Contact( #CIMCORP_MoveOK_P2 )
      Contact( #CIMCORP_OK )
      wire#w2
      Coil( #AVTF_Mx_MSig )
   END_RUNG
   RUNG wire#powerrail
      Contact( #Mx_ET50 )
   END_RUNG wire#w1
   RUNG wire#powerrail
      Contact( #Mx_ET51 )
      Contact( #EstadoVI.Descarga_Act )
   END_RUNG wire#w1
   RUNG wire#w2
      Coil( #STAT_AVTF_Mx_MSig )
   END_RUNG
   // the same network as SCL:
   #AVTF_Mx_MSig := ((#Mx_ET02 AND NOT #FTF_Mx_MSig AND #OrdSal_S03 AND NOT #EstadoZona.ParoBlando_CBx) OR #Mx_ET50 OR (#Mx_ET51 AND #EstadoVI.Descarga_Act)) AND #EstadoZona.Marcha_CBx AND NOT #Error_Tx AND #CIMCORP_MoveOK_P1 AND #CIMCORP_MoveOK_P2 AND #CIMCORP_OK;
   #STAT_AVTF_Mx_MSig := #AVTF_Mx_MSig;
END_REGION

REGION Network 40: VARIABLES AUXILIARES - P_Mens_Mx_MSig (Nota: solo en ET51)
   RUNG wire#powerrail
      Contact( #Mx_ET51 )
      wire#w1
      Coil( #P_Mens_Mx_MSig )
   END_RUNG
   RUNG wire#powerrail
      Contact( #Mx_ET50 )
      { S7_Templates := "SrcType := Int" } GE_Contact(in1 := #CNTSeg_ApHsMx.CVU, in2 := #V_CNTSeg_ApHsMx)
      Contact( "OFF" )
   END_RUNG wire#w1
   // the same network as SCL:
   #P_Mens_Mx_MSig := #Mx_ET51 OR (#Mx_ET50 AND (#CNTSeg_ApHsMx.CVU >= #V_CNTSeg_ApHsMx) AND "OFF");
END_REGION

REGION Network 41: MENSAJES - PRESENCIA
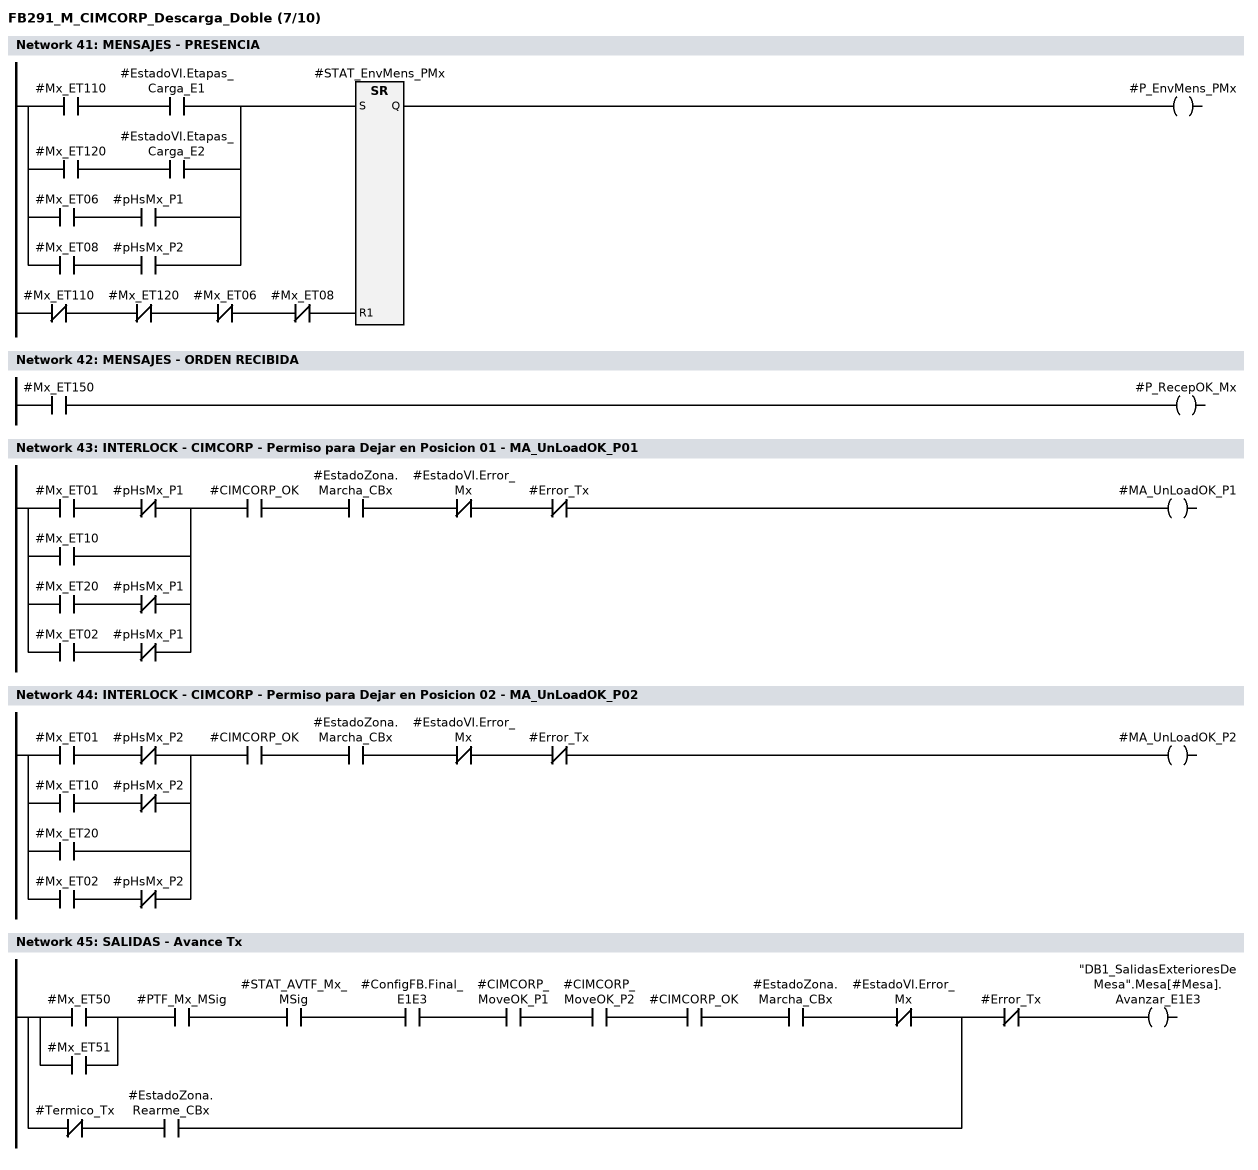
   RUNG wire#powerrail
      Contact( #Mx_ET110 )
      Contact( #EstadoVI.Etapas_Carga_E1 )
      wire#w1
      S_SR(operand := #STAT_EnvMens_PMx, r1 := wire#w2)
      Coil( #P_EnvMens_PMx )
   END_RUNG
   RUNG wire#powerrail
      Contact( #Mx_ET120 )
      Contact( #EstadoVI.Etapas_Carga_E2 )
   END_RUNG wire#w1
   RUNG wire#powerrail
      Contact( #Mx_ET06 )
      Contact( #pHsMx_P1 )
   END_RUNG wire#w1
   RUNG wire#powerrail
      Contact( #Mx_ET08 )
      Contact( #pHsMx_P2 )
   END_RUNG wire#w1
   RUNG wire#powerrail
      I_Contact( #Mx_ET110 )
      I_Contact( #Mx_ET120 )
      I_Contact( #Mx_ET06 )
      I_Contact( #Mx_ET08 )
   END_RUNG wire#w2
   // the same network as SCL:
   IF (#Mx_ET110 AND #EstadoVI.Etapas_Carga_E1) OR (#Mx_ET120 AND #EstadoVI.Etapas_Carga_E2) OR (#Mx_ET06 AND #pHsMx_P1) OR (#Mx_ET08 AND #pHsMx_P2) THEN
       #STAT_EnvMens_PMx := TRUE;   // SR flip-flop
   END_IF;
   IF NOT #Mx_ET110 AND NOT #Mx_ET120 AND NOT #Mx_ET06 AND NOT #Mx_ET08 THEN
       #STAT_EnvMens_PMx := FALSE;
   END_IF;
   #P_EnvMens_PMx := #STAT_EnvMens_PMx;
END_REGION

REGION Network 42: MENSAJES - ORDEN RECIBIDA
   RUNG wire#powerrail
      Contact( #Mx_ET150 )
      Coil( #P_RecepOK_Mx )
   END_RUNG
   // the same network as SCL:
   #P_RecepOK_Mx := #Mx_ET150;
END_REGION

REGION Network 43: INTERLOCK - CIMCORP - Permiso para Dejar en Posicion 01 - MA_UnLoadOK_P01
   RUNG wire#powerrail
      Contact( #Mx_ET01 )
      I_Contact( #pHsMx_P1 )
      wire#w1
      Contact( #CIMCORP_OK )
      Contact( #EstadoZona.Marcha_CBx )
      I_Contact( #EstadoVI.Error_Mx )
      I_Contact( #Error_Tx )
      Coil( #MA_UnLoadOK_P1 )
   END_RUNG
   RUNG wire#powerrail
      Contact( #Mx_ET10 )
   END_RUNG wire#w1
   RUNG wire#powerrail
      Contact( #Mx_ET20 )
      I_Contact( #pHsMx_P1 )
   END_RUNG wire#w1
   RUNG wire#powerrail
      Contact( #Mx_ET02 )
      I_Contact( #pHsMx_P1 )
   END_RUNG wire#w1
   // the same network as SCL:
   #MA_UnLoadOK_P1 := ((#Mx_ET01 AND NOT #pHsMx_P1) OR #Mx_ET10 OR (#Mx_ET20 AND NOT #pHsMx_P1) OR (#Mx_ET02 AND NOT #pHsMx_P1)) AND #CIMCORP_OK AND #EstadoZona.Marcha_CBx AND NOT #EstadoVI.Error_Mx AND NOT #Error_Tx;
END_REGION

REGION Network 44: INTERLOCK - CIMCORP - Permiso para Dejar en Posicion 02 - MA_UnLoadOK_P02
   RUNG wire#powerrail
      Contact( #Mx_ET01 )
      I_Contact( #pHsMx_P2 )
      wire#w1
      Contact( #CIMCORP_OK )
      Contact( #EstadoZona.Marcha_CBx )
      I_Contact( #EstadoVI.Error_Mx )
      I_Contact( #Error_Tx )
      Coil( #MA_UnLoadOK_P2 )
   END_RUNG
   RUNG wire#powerrail
      Contact( #Mx_ET10 )
      I_Contact( #pHsMx_P2 )
   END_RUNG wire#w1
   RUNG wire#powerrail
      Contact( #Mx_ET20 )
   END_RUNG wire#w1
   RUNG wire#powerrail
      Contact( #Mx_ET02 )
      I_Contact( #pHsMx_P2 )
   END_RUNG wire#w1
   // the same network as SCL:
   #MA_UnLoadOK_P2 := ((#Mx_ET01 AND NOT #pHsMx_P2) OR (#Mx_ET10 AND NOT #pHsMx_P2) OR #Mx_ET20 OR (#Mx_ET02 AND NOT #pHsMx_P2)) AND #CIMCORP_OK AND #EstadoZona.Marcha_CBx AND NOT #EstadoVI.Error_Mx AND NOT #Error_Tx;
END_REGION

REGION Network 45: SALIDAS - Avance Tx
   RUNG wire#powerrail
      Contact( #Mx_ET50 )
      wire#w1
      Contact( #PTF_Mx_MSig )
      Contact( #STAT_AVTF_Mx_MSig )
      Contact( #ConfigFB.Final_E1E3 )
      Contact( #CIMCORP_MoveOK_P1 )
      Contact( #CIMCORP_MoveOK_P2 )
      Contact( #CIMCORP_OK )
      Contact( #EstadoZona.Marcha_CBx )
      I_Contact( #EstadoVI.Error_Mx )
      wire#w2
      I_Contact( #Error_Tx )
      Coil( "DB1_SalidasExterioresDeMesa".Mesa[#Mesa].Avanzar_E1E3 )
   END_RUNG
   RUNG wire#powerrail
      Contact( #Mx_ET51 )
   END_RUNG wire#w1
   RUNG wire#powerrail
      I_Contact( #Termico_Tx )
      Contact( #EstadoZona.Rearme_CBx )
   END_RUNG wire#w2
   // the same network as SCL:
   "DB1_SalidasExterioresDeMesa".Mesa[#Mesa].Avanzar_E1E3 := (((#Mx_ET50 OR #Mx_ET51) AND #PTF_Mx_MSig AND #STAT_AVTF_Mx_MSig AND #ConfigFB.Final_E1E3 AND #CIMCORP_MoveOK_P1 AND #CIMCORP_MoveOK_P2 AND #CIMCORP_OK AND #EstadoZona.Marcha_CBx AND NOT #EstadoVI.Error_Mx) OR (NOT #Termico_Tx AND #EstadoZona.Rearme_CBx)) AND NOT #Error_Tx;
END_REGION

REGION Network 46: SALIDAS - Parar Tx
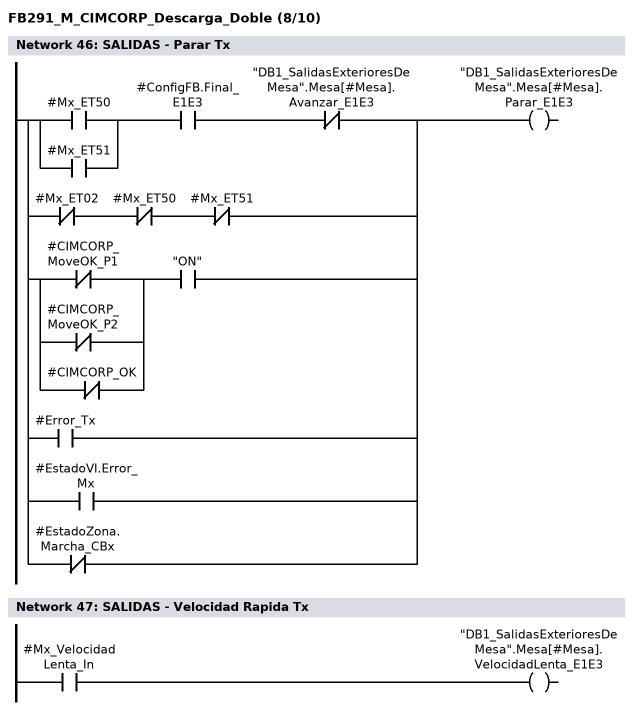
   RUNG wire#powerrail
      Contact( #Mx_ET50 )
      wire#w1
      Contact( #ConfigFB.Final_E1E3 )
      I_Contact( "DB1_SalidasExterioresDeMesa".Mesa[#Mesa].Avanzar_E1E3 )
      wire#w2
      Coil( "DB1_SalidasExterioresDeMesa".Mesa[#Mesa].Parar_E1E3 )
   END_RUNG
   RUNG wire#powerrail
      Contact( #Mx_ET51 )
   END_RUNG wire#w1
   RUNG wire#powerrail
      I_Contact( #Mx_ET02 )
      I_Contact( #Mx_ET50 )
      I_Contact( #Mx_ET51 )
   END_RUNG wire#w2
   RUNG wire#powerrail
      I_Contact( #CIMCORP_MoveOK_P1 )
      wire#w3
      Contact( "ON" )
   END_RUNG wire#w2
   RUNG wire#powerrail
      I_Contact( #CIMCORP_MoveOK_P2 )
   END_RUNG wire#w3
   RUNG wire#powerrail
      I_Contact( #CIMCORP_OK )
   END_RUNG wire#w3
   RUNG wire#powerrail
      Contact( #Error_Tx )
   END_RUNG wire#w2
   RUNG wire#powerrail
      Contact( #EstadoVI.Error_Mx )
   END_RUNG wire#w2
   RUNG wire#powerrail
      I_Contact( #EstadoZona.Marcha_CBx )
   END_RUNG wire#w2
   // the same network as SCL:
   "DB1_SalidasExterioresDeMesa".Mesa[#Mesa].Parar_E1E3 := ((#Mx_ET50 OR #Mx_ET51) AND #ConfigFB.Final_E1E3 AND NOT "DB1_SalidasExterioresDeMesa".Mesa[#Mesa].Avanzar_E1E3) OR (NOT #Mx_ET02 AND NOT #Mx_ET50 AND NOT #Mx_ET51) OR ((NOT #CIMCORP_MoveOK_P1 OR NOT #CIMCORP_MoveOK_P2 OR NOT #CIMCORP_OK) AND "ON") OR #Error_Tx OR #EstadoVI.Error_Mx OR NOT #EstadoZona.Marcha_CBx;
END_REGION

REGION Network 47: SALIDAS - Velocidad Rapida Tx
   RUNG wire#powerrail
      Contact( #Mx_VelocidadLenta_In )
      Coil( "DB1_SalidasExterioresDeMesa".Mesa[#Mesa].VelocidadLenta_E1E3 )
   END_RUNG
   // the same network as SCL:
   "DB1_SalidasExterioresDeMesa".Mesa[#Mesa].VelocidadLenta_E1E3 := #Mx_VelocidadLenta_In;
END_REGION

REGION Network 48: ESTADOS DE LA MESA
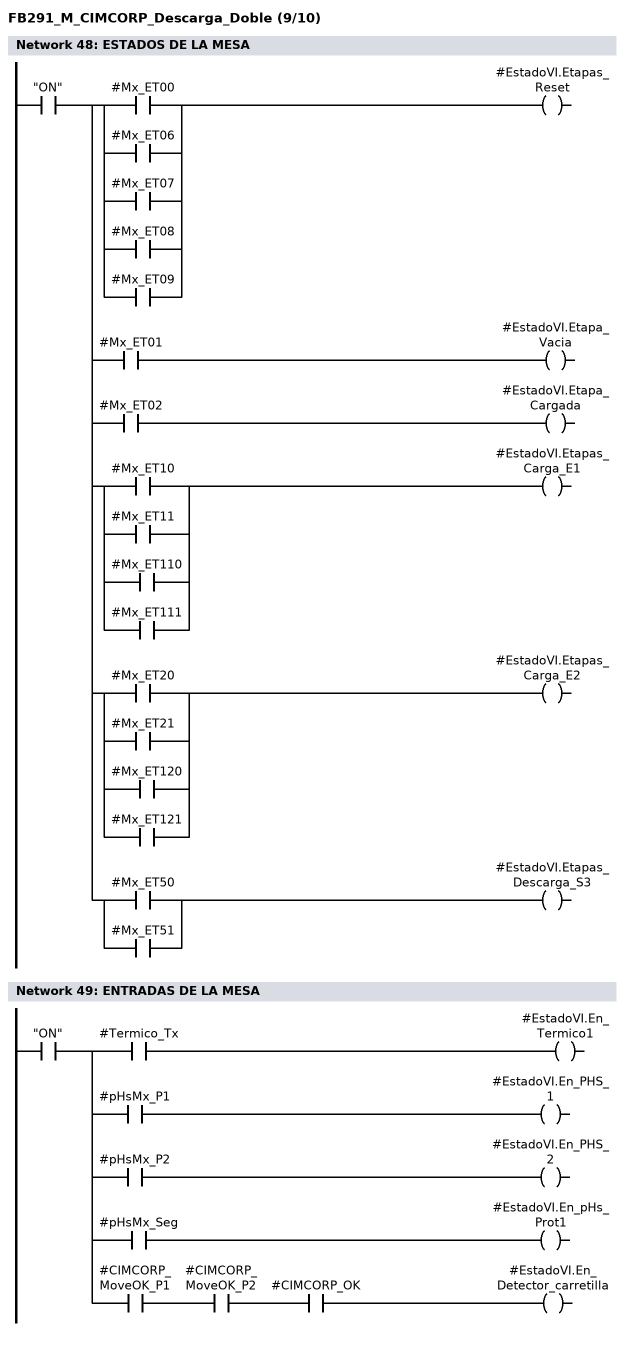
   RUNG wire#powerrail
      Contact( "ON" )
      wire#w1
      Contact( #Mx_ET00 )
      wire#w2
      Coil( #EstadoVI.Etapas_Reset )
   END_RUNG
   RUNG wire#w1
      Contact( #Mx_ET06 )
   END_RUNG wire#w2
   RUNG wire#w1
      Contact( #Mx_ET07 )
   END_RUNG wire#w2
   RUNG wire#w1
      Contact( #Mx_ET08 )
   END_RUNG wire#w2
   RUNG wire#w1
      Contact( #Mx_ET09 )
   END_RUNG wire#w2
   RUNG wire#w1
      Contact( #Mx_ET01 )
      Coil( #EstadoVI.Etapa_Vacia )
   END_RUNG
   RUNG wire#w1
      Contact( #Mx_ET02 )
      Coil( #EstadoVI.Etapa_Cargada )
   END_RUNG
   RUNG wire#w1
      Contact( #Mx_ET10 )
      wire#w3
      Coil( #EstadoVI.Etapas_Carga_E1 )
   END_RUNG
   RUNG wire#w1
      Contact( #Mx_ET11 )
   END_RUNG wire#w3
   RUNG wire#w1
      Contact( #Mx_ET110 )
   END_RUNG wire#w3
   RUNG wire#w1
      Contact( #Mx_ET111 )
   END_RUNG wire#w3
   RUNG wire#w1
      Contact( #Mx_ET20 )
      wire#w4
      Coil( #EstadoVI.Etapas_Carga_E2 )
   END_RUNG
   RUNG wire#w1
      Contact( #Mx_ET21 )
   END_RUNG wire#w4
   RUNG wire#w1
      Contact( #Mx_ET120 )
   END_RUNG wire#w4
   RUNG wire#w1
      Contact( #Mx_ET121 )
   END_RUNG wire#w4
   RUNG wire#w1
      Contact( #Mx_ET50 )
      wire#w5
      Coil( #EstadoVI.Etapas_Descarga_S3 )
   END_RUNG
   RUNG wire#w1
      Contact( #Mx_ET51 )
   END_RUNG wire#w5
   // the same network as SCL:
   #EstadoVI.Etapas_Reset := "ON" AND (#Mx_ET00 OR #Mx_ET06 OR #Mx_ET07 OR #Mx_ET08 OR #Mx_ET09);
   #EstadoVI.Etapa_Vacia := "ON" AND #Mx_ET01;
   #EstadoVI.Etapa_Cargada := "ON" AND #Mx_ET02;
   #EstadoVI.Etapas_Carga_E1 := "ON" AND (#Mx_ET10 OR #Mx_ET11 OR #Mx_ET110 OR #Mx_ET111);
   #EstadoVI.Etapas_Carga_E2 := "ON" AND (#Mx_ET20 OR #Mx_ET21 OR #Mx_ET120 OR #Mx_ET121);
   #EstadoVI.Etapas_Descarga_S3 := "ON" AND (#Mx_ET50 OR #Mx_ET51);
END_REGION

REGION Network 49: ENTRADAS DE LA MESA
   RUNG wire#powerrail
      Contact( "ON" )
      wire#w1
      Contact( #Termico_Tx )
      Coil( #EstadoVI.En_Termico1 )
   END_RUNG
   RUNG wire#w1
      Contact( #pHsMx_P1 )
      Coil( #EstadoVI.En_PHS_1 )
   END_RUNG
   RUNG wire#w1
      Contact( #pHsMx_P2 )
      Coil( #EstadoVI.En_PHS_2 )
   END_RUNG
   RUNG wire#w1
      Contact( #pHsMx_Seg )
      Coil( #EstadoVI.En_pHs_Prot1 )
   END_RUNG
   RUNG wire#w1
      Contact( #CIMCORP_MoveOK_P1 )
      Contact( #CIMCORP_MoveOK_P2 )
      Contact( #CIMCORP_OK )
      Coil( #EstadoVI.En_Detector_carretilla )
   END_RUNG
   // the same network as SCL:
   #EstadoVI.En_Termico1 := "ON" AND #Termico_Tx;
   #EstadoVI.En_PHS_1 := "ON" AND #pHsMx_P1;
   #EstadoVI.En_PHS_2 := "ON" AND #pHsMx_P2;
   #EstadoVI.En_pHs_Prot1 := "ON" AND #pHsMx_Seg;
   #EstadoVI.En_Detector_carretilla := "ON" AND #CIMCORP_MoveOK_P1 AND #CIMCORP_MoveOK_P2 AND #CIMCORP_OK;
END_REGION

REGION Network 50: SALIDAS DE LA MESA
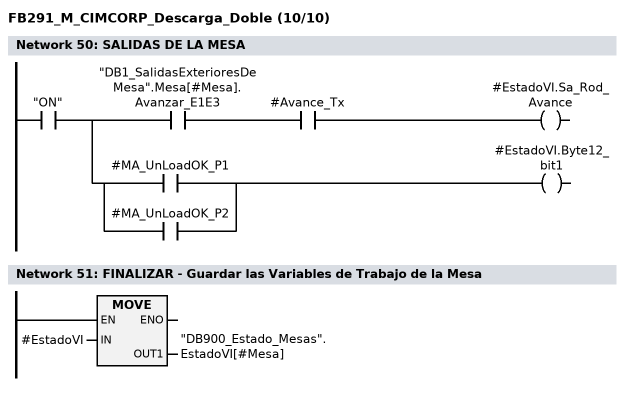
   RUNG wire#powerrail
      Contact( "ON" )
      wire#w1
      Contact( "DB1_SalidasExterioresDeMesa".Mesa[#Mesa].Avanzar_E1E3 )
      Contact( #Avance_Tx )
      Coil( #EstadoVI.Sa_Rod_Avance )
   END_RUNG
   RUNG wire#w1
      Contact( #MA_UnLoadOK_P1 )
      wire#w2
      Coil( #EstadoVI.Byte12_bit1 )
   END_RUNG
   RUNG wire#w1
      Contact( #MA_UnLoadOK_P2 )
   END_RUNG wire#w2
   // the same network as SCL:
   #EstadoVI.Sa_Rod_Avance := "ON" AND "DB1_SalidasExterioresDeMesa".Mesa[#Mesa].Avanzar_E1E3 AND #Avance_Tx;
   #EstadoVI.Byte12_bit1 := "ON" AND (#MA_UnLoadOK_P1 OR #MA_UnLoadOK_P2);
END_REGION

REGION Network 51: FINALIZAR - Guardar las Variables de Trabajo de la Mesa
   RUNG wire#powerrail
      Move(in := #EstadoVI, out1 => "DB900_Estado_Mesas".EstadoVI[#Mesa])
   END_RUNG
   // the same network as SCL:
   "DB900_Estado_Mesas".EstadoVI[#Mesa] := #EstadoVI;
END_REGION
END_FUNCTION_BLOCK
